TYPE ST_AXIS_VEL_STATUS :
STRUCT
END_STRUCT
END_TYPE

(* stored: Version 1.1.0.1, ProductVersion 3.1.4024.11
   DUT ST_AXIS_VEL_STATUS: Id {37451264-81f5-45ce-9096-4c211dce929f} *)
